TYPE XTSMainControl_typ :
STRUCT
Cmd	: XTSMainCommands_typ;
Sts	: XTSMainStatus_typ;
END_STRUCT
END_TYPE

(* stored: Version 1.1.0.1, ProductVersion 3.1.4024.12
   DUT XTSMainControl_typ: Id {cc226de0-506d-0290-3d19-003bad9e801e} *)
